// TIA Portal V20 export
TYPE "LKinCtrl_typeExecuteKinMotionCmdDiagnostics"
   STRUCT
      status : Word;   // status of the FB
      faultPathDataName : String["LKINCTRL_LENGTH_OF_PATHDATA_NAME"];   // number of PathData with occurring error in PathData set
      faultSetNumber : DInt;   // number of PathData set with occurring error
      faultFBNumber : DInt;   // number of motionCommand FB with occurring error
      motionFBstatus : DWord;   // status of motion FB (internal) an error occurred in
      stateMachine : Int;   // stateMachine status
      kinematicsStatusWord : DWord;   // statusWord TO kinematics
      kinematicsErrorWord : DWord;   // errorWord TO kinematics
   END_STRUCT;
END_TYPE
